(* PLC project bottling_line, Dassault Systèmes ControlBuild 2024x *)
(* stored: creationDateTime 2023-10-05T15:43:44-01:00 *)

CONFIGURATION bottling_line
  VAR_GLOBAL
    simuperiod : REAL := 50000.0;
    taskname : STRING(50) := 'bottling_line.exe';
    allowpreconditions : BOOL := true;
    allowpostconditions : BOOL := true;
    generalPanel/emergencyStopPB/PBLogic : BOOL := false;
    pumpingTank1/filling/inputFlow : REAL := 1000.0;
    pumpingTank1/filling/valve/flowMax : REAL := 1000.0;
    pumpingTank1/filling/valve/flowPerHour : BOOL := false;
    pumpingTank1/filling/valve/flowPerMinute : BOOL := true;
    pumpingTank1/emptying/valve/flowMax : REAL := 1000.0;
    pumpingTank1/emptying/valve/flowPerHour : BOOL := false;
    pumpingTank1/emptying/valve/flowPerMinute : BOOL := true;
    pumpingTank1/tank/capacity : REAL := 500.0;
    pumpingTank1/extraction/pump/flowMax : REAL := 1000.0;
    pumpingTank1/extraction/pump/flowPerHour : BOOL := false;
    pumpingTank1/extraction/pump/flowPerMinute : BOOL := true;
    pumpingTank1/levelScale/maxInput : REAL := 500.0;
    pumpingTank1/highLevel/threshold : REAL := 490.0;
    pumpingTank1/lowLevel/threshold : REAL := 30.0;
    pumpingTank1/lowLevel/wiringLogic : BOOL := false;
    pumpingTank2/filling/inputFlow : REAL := 1000.0;
    pumpingTank2/filling/valve/flowMax : REAL := 1000.0;
    pumpingTank2/filling/valve/flowPerHour : BOOL := false;
    pumpingTank2/filling/valve/flowPerMinute : BOOL := true;
    pumpingTank2/emptying/valve/flowMax : REAL := 1000.0;
    pumpingTank2/emptying/valve/flowPerHour : BOOL := false;
    pumpingTank2/emptying/valve/flowPerMinute : BOOL := true;
    pumpingTank2/tank/capacity : REAL := 500.0;
    pumpingTank2/extraction/pump/flowMax : REAL := 1000.0;
    pumpingTank2/extraction/pump/flowPerHour : BOOL := false;
    pumpingTank2/extraction/pump/flowPerMinute : BOOL := true;
    pumpingTank2/levelScale/maxInput : REAL := 500.0;
    pumpingTank2/highLevel/threshold : REAL := 490.0;
    pumpingTank2/lowLevel/threshold : REAL := 30.0;
    pumpingTank2/lowLevel/wiringLogic : BOOL := false;
    mixing/flow/flowMax : REAL := 2000.0;
    mixing/flow/flowPerHour : BOOL := false;
    mixing/flow/flowPerMinute : BOOL := true;
    mixing/valve5/valve/flowMax : REAL := 100000.0;
    mixing/valve5/valve/flowPerHour : BOOL := false;
    mixing/levelScale/maxInput : REAL := 1000.0;
    mixing/highLevel3/threshold : REAL := 950.0;
    mixing/lowLevel3/threshold : REAL := 100.0;
    mixing/lowLevel3/wiringLogic : BOOL := false;
    drive/pulse/pulseDuration : REAL := 0.3;
  END_VAR
END_CONFIGURATION
